PROGRAM SafetyInterface_Enc057
VAR
	{attribute 'TcLinkTo' := '
		.iSafteyCtrlProjectCRC := TIIB[N40S14 (EL6910)]^Device Info Data^Project CRC;
		.iSafetyGroup_State := TIIB[N40S14 (EL6910)]^TwinSAFE Group Info Data^Enc057_SafetyGroup Info Data^State;
		.iSafetyGroup_Diag := TIIB[N40S14 (EL6910)]^TwinSAFE Group Info Data^Enc057_SafetyGroup Info Data^Diag;
		.iSafetyGroup_ComErr := TIIB[N40S14 (EL6910)]^StandardInputs^Enc057_SafetyGroup.oGroup_ComErr_3;
		.iSafetyGroup_ComInStartup := TIIB[N40S14 (EL6910)]^StandardInputs^Enc057_SafetyGroup.oGroup_ComInStartup_4;
		.iSafetyGroup_FBErr := TIIB[N40S14 (EL6910)]^StandardInputs^Enc057_SafetyGroup.oGroup_FBErr_5;
		.iSafetyGroup_FBInRun := TIIB[N40S14 (EL6910)]^StandardInputs^Enc057_SafetyGroup.oGroup_FBInRun_6;
		.iSafetyGroup_InRun := TIIB[N40S14 (EL6910)]^StandardInputs^Enc057_SafetyGroup.oGroup_InRun_7;
		.iSafetyGroup_OtherErr := TIIB[N40S14 (EL6910)]^StandardInputs^Enc057_SafetyGroup.oGroup_OtherErr_8;
		.oSafetyGroup_ErrAck := TIIB[N40S14 (EL6910)]^StandardOutputs^Enc057_SafetyGroup.iGroup_ErrAck_1;
		.oSafetyGroup_Run := TIIB[N40S14 (EL6910)]^StandardOutputs^Enc057_SafetyGroup.iGroup_Run_2;
		.oControlPowerPBLight := TIIB[N40S09 (EL2008)]^Channel 1^Output;
		.iSafetyResetPB := TIIB[N40S14 (EL6910)]^Connection Info Data^Enc057_SafetyGroup.N40S01 Digital 4 In (EL1904)_9 Info Data^Input Safe Data InputChannel3;
		.iEstopPB1_CH1 := TIIB[N40S14 (EL6910)]^Connection Info Data^Enc057_SafetyGroup.N40S01 Digital 4 In (EL1904)_9 Info Data^Input Safe Data InputChannel1;
		.iEstopPB1_CH2 := TIIB[N40S14 (EL6910)]^Connection Info Data^Enc057_SafetyGroup.N40S01 Digital 4 In (EL1904)_9 Info Data^Input Safe Data InputChannel2;
		.iRelayNCContact_Estop := TIIB[N40S14 (EL6910)]^Connection Info Data^Enc057_SafetyGroup.N40S03 Digital 4 In (EL1904)_11 Info Data^Input Safe Data InputChannel1;
		.iSafetyPowerOn_Estop_CH1 := TIIB[N40S14 (EL6910)]^Connection Info Data^Enc057_SafetyGroup.N40S04 Digital 4 Out (EL2904)_20 Info Data^Output Safe Data OutputChannel1;
		.iSafetyPowerOn_Estop_CH2 := TIIB[N40S14 (EL6910)]^Connection Info Data^Enc057_SafetyGroup.N40S04 Digital 4 Out (EL2904)_20 Info Data^Output Safe Data OutputChannel2;
		.iAirPressureOk := TIIB[N40S06 (EL1008)]^Channel 2^Input'}
	fbSafetyInterface : FB_SafetyInterfaceConv;
END_VAR



fbSafetyInterface(
	pSafetyInterface := ADR(gProduced_SafetyInterfaceConv.Enc057));

END_PROGRAM

(* stored: Version 1.1.0.1, ProductVersion 3.1.4024.6
   POU SafetyInterface_Enc057: Id {7996bb58-4250-4897-a19c-a233ef203ed1}, SpecialFunc None *)
